FUNCTION_BLOCK Axis
VAR_INPUT
	execute:BOOL;
	pos :real;
	vel:INT;
	enable : BOOL;
	reset : BOOL;
END_VAR
VAR_OUTPUT
END_VAR
VAR
	axis: AXIS_REF;
	moveabs: MC_moveabsolute;
	power : MC_power;
	resetaxis: MC_reset;
	
END_VAR

power(axis:=axis);
moveabs(axis:=axis);
resetaxis(axis := axis);
power.Enable := enable;

resetaxis.execute := reset;
power.Enable_Negative:= TRUE;
power.Enable_Positive:= TRUE;
moveabs.Velocity := vel;
moveabs.Position := pos;
moveabs.Execute := execute;

END_FUNCTION_BLOCK

(* stored: Version 1.1.0.1, ProductVersion 3.1.4024.12
   POU Axis: Id {fad8b9b6-b69e-4ba0-adbe-b22ee12d4b8e}, SpecialFunc None *)
